(* CoDeSys 2.3.9.41 project: fongus.pro *)
(* Libraries: STANDARD.LIB 4.10.05 11:14:46, IECSFC.LIB 13.4.06 15:51:28, ANALYZATION.LIB 5.10.99 09:05:06 *)

(* PLC configuration (modules and I/O channels)
DI0_staticRun AT %IX0.0 [BitInput]
DI1_dynamicRun AT %IX0.1 [BitInput]
AT %IX0.2 [BitInput]
AT %IX0.3 [BitInput]
AT %IX0.4 [BitInput]
AT %IX0.5 [BitInput]
DO0_filter AT %QX1.0 [BitOutput]
AT %QX1.1 [BitOutput]
AT %QX1.2 [BitOutput]
AT %QX1.3 [BitOutput]
Special output [ID104] node 2, in %IB2 out %QB2 {Visibility = No; PinCount = 1}
  AT %QX2.0 [BitOutput] Special output
Unifed signal sensor [ID700] node 3, in %IB3 out %QB3 {Type_of_sensor700 = IT_0_20; measure_interval = 0.8; ainlow = 0; ainhigh = 20; first_cor_point = 0; first_delta = 0; second_cor_point = 0; second_delta = 0; third_cor_point = 0; third_delta = 0; Visibility = No}
  AT %ID3.0 [FloatInput] Value
  AT %IW3.1 [WordInput] Circular time
  Analog Input [ID107] node 0, in %IB3.0 out %QB3.0
Unifed signal sensor [ID700] node 4, in %IB4 out %QB4 {Type_of_sensor700 = IT_0_20; measure_interval = 0.8; ainlow = 0; ainhigh = 20; first_cor_point = 0; first_delta = 0; second_cor_point = 0; second_delta = 0; third_cor_point = 0; third_delta = 0; Visibility = No}
  AT %ID4.0 [FloatInput] Value
  AT %IW4.1 [WordInput] Circular time
  Analog Input [ID107] node 0, in %IB4.0 out %QB4.0
Unifed signal sensor [ID700] node 5, in %IB5 out %QB5 {Type_of_sensor700 = IT_0_20; measure_interval = 0.8; ainlow = 0; ainhigh = 20; first_cor_point = 0; first_delta = 0; second_cor_point = 0; second_delta = 0; third_cor_point = 0; third_delta = 0; Visibility = No}
  AT %ID5.0 [FloatInput] Value
  AT %IW5.1 [WordInput] Circular time
  Analog Input [ID107] node 0, in %IB5.0 out %QB5.0
Unifed signal sensor [ID700] node 6, in %IB6 out %QB6 {Type_of_sensor700 = IT_0_20; measure_interval = 0.8; ainlow = 0; ainhigh = 20; first_cor_point = 0; first_delta = 0; second_cor_point = 0; second_delta = 0; third_cor_point = 0; third_delta = 0; Visibility = No}
  AT %ID6.0 [FloatInput] Value
  AT %IW6.1 [WordInput] Circular time
  Analog Input [ID107] node 0, in %IB6.0 out %QB6.0
AO0_fc1 AT %QD7.0 [FloatOutput] Value
AO1_fc2 AT %QD8.0 [FloatOutput] Value
Modbus [MODBUS_ID302] node 0, in %IB9.0 out %QB9.0
  Debug RS-232 [DEBUG_USART] node 0, in %IB9.0.0 out %QB9.0.0 {CommunicationSpeed = 11520; Parity = NO PARITY CHECK; BitLength = 8 bits; StopLength = One stop bit; InterfaceType = RS232; FrameOriented = ASCII; Timeout = 0; Visibility = No}
pan_BITS0 AT %QW9.1.0 [WordOutput] man
pan_BITS1 AT %QW9.2.0 [WordOutput]
pan_BITS2 AT %QW9.3.0 [WordOutput]
pan_BITS3 AT %QW9.4.0 [WordOutput]
2 byte [Register] node 5, in %IB9.5 out %QB9.5
  fc1_p1t AT %QW9.5.0 [WordOutput]
2 byte [Register] node 6, in %IB9.6 out %QB9.6
  fc1_p2t AT %QW9.6.0 [WordOutput]
2 byte [Register] node 7, in %IB9.7 out %QB9.7
  fc1_p3t AT %QW9.7.0 [WordOutput]
2 byte [Register] node 8, in %IB9.8 out %QB9.8
  fc1_p4t AT %QW9.8.0 [WordOutput]
2 byte [Register] node 9, in %IB9.9 out %QB9.9
  fc1_p5t AT %QW9.9.0 [WordOutput]
2 byte [Register] node 10, in %IB9.10 out %QB9.10
  fc1_p6t AT %QW9.10.0 [WordOutput]
2 byte [Register] node 11, in %IB9.11 out %QB9.11
  fc1_p7t AT %QW9.11.0 [WordOutput]
2 byte [Register] node 12, in %IB9.12 out %QB9.12
  fc1_p8t AT %QW9.12.0 [WordOutput]
2 byte [Register] node 13, in %IB9.13 out %QB9.13
  fc1_p9t AT %QW9.13.0 [WordOutput]
2 byte [Register] node 14, in %IB9.14 out %QB9.14
  fc1_p10t AT %QW9.14.0 [WordOutput]
2 byte [Register] node 15, in %IB9.15 out %QB9.15
  fc1_p1v AT %QW9.15.0 [WordOutput]
2 byte [Register] node 16, in %IB9.16 out %QB9.16
  fc1_p2v AT %QW9.16.0 [WordOutput]
2 byte [Register] node 17, in %IB9.17 out %QB9.17
  fc1_p3v AT %QW9.17.0 [WordOutput]
2 byte [Register] node 18, in %IB9.18 out %QB9.18
  fc1_p4v AT %QW9.18.0 [WordOutput]
2 byte [Register] node 19, in %IB9.19 out %QB9.19
  fc1_p5v AT %QW9.19.0 [WordOutput]
2 byte [Register] node 20, in %IB9.20 out %QB9.20
  fc1_p6v AT %QW9.20.0 [WordOutput]
2 byte [Register] node 21, in %IB9.21 out %QB9.21
  fc1_p7v AT %QW9.21.0 [WordOutput]
2 byte [Register] node 22, in %IB9.22 out %QB9.22
  fc1_p8v AT %QW9.22.0 [WordOutput]
2 byte [Register] node 23, in %IB9.23 out %QB9.23
  fc1_p9v AT %QW9.23.0 [WordOutput]
2 byte [Register] node 24, in %IB9.24 out %QB9.24
  fc1_p10v AT %QW9.24.0 [WordOutput]
2 byte [Register] node 25, in %IB9.25 out %QB9.25
  fc2_p1t AT %QW9.25.0 [WordOutput]
2 byte [Register] node 26, in %IB9.26 out %QB9.26
  fc2_p2t AT %QW9.26.0 [WordOutput]
2 byte [Register] node 27, in %IB9.27 out %QB9.27
  fc2_p3t AT %QW9.27.0 [WordOutput]
2 byte [Register] node 28, in %IB9.28 out %QB9.28
  fc2_p4t AT %QW9.28.0 [WordOutput]
2 byte [Register] node 29, in %IB9.29 out %QB9.29
  fc2_p5t AT %QW9.29.0 [WordOutput]
2 byte [Register] node 30, in %IB9.30 out %QB9.30
  fc2_p6t AT %QW9.30.0 [WordOutput]
2 byte [Register] node 31, in %IB9.31 out %QB9.31
  fc2_p7t AT %QW9.31.0 [WordOutput]
2 byte [Register] node 32, in %IB9.32 out %QB9.32
  fc2_p8t AT %QW9.32.0 [WordOutput]
2 byte [Register] node 33, in %IB9.33 out %QB9.33
  fc2_p9t AT %QW9.33.0 [WordOutput]
2 byte [Register] node 34, in %IB9.34 out %QB9.34
  fc2_p10t AT %QW9.34.0 [WordOutput]
2 byte [Register] node 35, in %IB9.35 out %QB9.35
  fc2_p1v AT %QW9.35.0 [WordOutput]
2 byte [Register] node 36, in %IB9.36 out %QB9.36
  fc2_p2v AT %QW9.36.0 [WordOutput]
2 byte [Register] node 37, in %IB9.37 out %QB9.37
  fc2_p3v AT %QW9.37.0 [WordOutput]
2 byte [Register] node 38, in %IB9.38 out %QB9.38
  fc2_p4v AT %QW9.38.0 [WordOutput]
2 byte [Register] node 39, in %IB9.39 out %QB9.39
  fc2_p5v AT %QW9.39.0 [WordOutput]
2 byte [Register] node 40, in %IB9.40 out %QB9.40
  fc2_p6v AT %QW9.40.0 [WordOutput]
2 byte [Register] node 41, in %IB9.41 out %QB9.41
  fc2_p7v AT %QW9.41.0 [WordOutput]
2 byte [Register] node 42, in %IB9.42 out %QB9.42
  fc2_p8v AT %QW9.42.0 [WordOutput]
2 byte [Register] node 43, in %IB9.43 out %QB9.43
  fc2_p9v AT %QW9.43.0 [WordOutput]
2 byte [Register] node 44, in %IB9.44 out %QB9.44
  fc2_p10v AT %QW9.44.0 [WordOutput]
2 byte [Register] node 45, in %IB9.45 out %QB9.45
  fc1_staticValue AT %QW9.45.0 [WordOutput]
  fc2_staticValue AT %QW9.46.0 [WordOutput]
  pan_evilStartHH AT %QW9.47.0 [WordOutput]
  pan_evilStartMM AT %QW9.48.0 [WordOutput]
  pan_evilStopHH AT %QW9.49.0 [WordOutput]
  pan_evilStopMM AT %QW9.50.0 [WordOutput]
  pan_holyStartHH AT %QW9.51.0 [WordOutput]
  pan_holyStartMM AT %QW9.52.0 [WordOutput]
  pan_holyStopHH AT %QW9.53.0 [WordOutput]
  pan_holyStopMM AT %QW9.54.0 [WordOutput]
  pan_EVILDAYS AT %QW9.55.0 [WordOutput]
  pan_HOLYDAYS AT %QW9.56.0 [WordOutput]
  pan_fe1_onHH AT %QW9.57.0 [WordOutput]
  pan_fe1_onMM AT %QW9.58.0 [WordOutput]
  pan_fe1_offHH AT %QW9.59.0 [WordOutput]
  pan_fe1_offMM AT %QW9.60.0 [WordOutput]
  pan_fe2_onHH AT %QW9.61.0 [WordOutput]
  pan_fe2_onMM AT %QW9.62.0 [WordOutput]
  pan_fe2_offHH AT %QW9.63.0 [WordOutput]
  pan_fe2_offMM AT %QW9.64.0 [WordOutput]
  pan_fe3_onHH AT %QW9.65.0 [WordOutput]
  pan_fe3_onMM AT %QW9.66.0 [WordOutput]
  pan_fe3_offHH AT %QW9.67.0 [WordOutput]
  pan_fe3_offMM AT %QW9.68.0 [WordOutput]
  pan_fe4_onHH AT %QW9.69.0 [WordOutput]
  pan_fe4_onMM AT %QW9.70.0 [WordOutput]
  pan_fe4_offHH AT %QW9.71.0 [WordOutput]
  pan_fe4_offMM AT %QW9.72.0 [WordOutput]
  pan_fe5_onHH AT %QW9.73.0 [WordOutput]
  pan_fe5_onMM AT %QW9.74.0 [WordOutput]
  pan_fe5_offHH AT %QW9.75.0 [WordOutput]
  pan_fe5_offMM AT %QW9.76.0 [WordOutput]
  pan_fe6_onHH AT %QW9.77.0 [WordOutput]
  pan_fe6_onMM AT %QW9.78.0 [WordOutput]
  pan_fe6_offHH AT %QW9.79.0 [WordOutput]
  pan_fe6_offMM AT %QW9.80.0 [WordOutput]
*)

(* Global variable list: Global_Variables *)
VAR_GLOBAL

(* Times *)
	GetTime: CurTimeEx;
	TimeAndDate: SystemTimeDate;
	Sys_Time: SysTime64;

END_VAR

(* POU PLC_PRG, ST *)
PROGRAM PLC_PRG
VAR
	setYear : INT;
	setMonth, setDay, setHour, setMinute : BYTE;
	set_time : BOOL;
END_VAR

END_PROGRAM
ACTION Times:
TimeAndDate.Day :=0;
TimeAndDate.DayOfWeek :=0;
TimeAndDate.dwHighMsec :=0;
TimeAndDate.dwLowMSecs :=0;
TimeAndDate.Milliseconds :=0;
TimeAndDate.Minute :=0;
TimeAndDate.Second :=0;
TimeAndDate.Hour :=0;
TimeAndDate.Year :=0;
TimeAndDate.Month :=0;
Sys_time.ulHigh :=0;
Sys_time.ulLow :=0;
GetTime (SystemTime:=Sys_Time , TimeDate:= TimeAndDate);


IF set_time THEN

	TimeAndDate.Minute:=setMinute;
	TimeAndDate.Second:=0;
	TimeAndDate.Hour:=setHour;
	TimeAndDate.Day:=setDay;
	TimeAndDate.Month:=setMonth;
	TimeAndDate.Year:=setYear;
	GetTime (SystemTime:=Sys_Time , TimeDate:= TimeAndDate);

END_IF
END_ACTION

(* POU FOUNTAIN, ST *)
PROGRAM FOUNTAIN
VAR
	start : BOOL;
	startByDays : BOOL;
	dynamic, static : BOOL;
	evilStartHH, evilStartMM, evilStopHH, evilStopMM : WORD;
	holyStartHH, holyStartMM, holyStopHH, holyStopMM : WORD;

	(* filter *)
	 filterRun, filterSchedGo : BOOL;
	fe1, fe2, fe3, fe4, fe5, fe6 : TimeOnCheck;
	fe1state, fe2state, fe3state, fe4state, fe5state, fe6state : BOOL;

	(* days *)
	evilTimeCheck, holyTimeCheck : TimeOnCheck;
	evilDayOk, holyDayOk : BOOL;

	M1, N1 : BOOL;
	founT1, founTN1 : TON;
	M2, N2 : BOOL;
	founT2, founTN2 : TON;
	M3, N3 : BOOL;
	founT3, founTN3 : TON;
	M4, N4 : BOOL;
	founT4, founTN4 : TON;
	M5, N5 : BOOL;
	founT5, founTN5 : TON;
	M6, N6 : BOOL;
	founT6, founTN6 : TON;
	M7, N7 : BOOL;
	founT7, founTN7 : TON;
	M8, N8 : BOOL;
	founT8, founTN8 : TON;
	M9, N9 : BOOL;
	founT9, founTN9 : TON;
	M10, N10 : BOOL;
	founT10, founTN10 : TON;

	FPFON: R_TRIG;
	FPFONN : R_TRIG;

	(*galetMode : BOOL;*)

END_VAR

VAR RETAIN
	(* filter *)
	filterMan, filterAuto : BOOL;
	fe1_onHH, fe1_onMM, fe1_offHH, fe1_offMM : WORD;
	fe2_onHH, fe2_onMM, fe2_offHH, fe2_offMM : WORD;
	fe3_onHH, fe3_onMM, fe3_offHH, fe3_offMM : WORD;
	fe4_onHH, fe4_onMM, fe4_offHH, fe4_offMM : WORD;
	fe5_onHH, fe5_onMM, fe5_offHH, fe5_offMM : WORD;
	fe6_onHH, fe6_onMM, fe6_offHH, fe6_offMM : WORD;

	staticFValue : REAL;
	staticFValueN : REAL;
	EVILDAYS, HOLYDAYS : WORD;

	(* fc1 *)
	founV1F: REAL;
	founV2F: REAL;
	founV3F: REAL;
	founV4F: REAL;
	founV5F: REAL;
	founV6F: REAL;
	founV7F: REAL;
	founV8F: REAL;
	founV9F: REAL;
	founV10F: REAL;

	founS1T: TIME;
	founS2T: TIME;
	founS3T: TIME;
	founS4T: TIME;
	founS5T: TIME;
	founS6T: TIME;
	founS7T: TIME;
	founS8T: TIME;
	founS9T: TIME;
	founS10T: TIME;

(* fc2 *)
	founV1FN: REAL;
	founV2FN: REAL;
	founV3FN: REAL;
	founV4FN: REAL;
	founV5FN: REAL;
	founV6FN: REAL;
	founV7FN: REAL;
	founV8FN: REAL;
	founV9FN: REAL;
	founV10FN: REAL;

	founS1TN: TIME;
	founS2TN: TIME;
	founS3TN: TIME;
	founS4TN: TIME;
	founS5TN: TIME;
	founS6TN: TIME;
	founS7TN: TIME;
	founS8TN: TIME;
	founS9TN: TIME;
	founS10TN: TIME;

(* days *)
	evilStartHH, evilStartMM, evilStopHH, evitStopMM : WORD;
	holyStartHH, holyStartMM, holyStopHH, holyStopMM : WORD;
END_VAR
VAR (* helpers for the ST form of the networks *)
	_p1 : BOOL;
	_p2 : BOOL;
	_p3 : BOOL;
	_p4 : BOOL;
	_p5 : BOOL;
	_p6 : BOOL;
	_p7 : BOOL;
	_p8 : BOOL;
	_p9 : BOOL;
	_p10 : BOOL;
	_p11 : BOOL;
	_p12 : BOOL;
	_p13 : BOOL;
	_p14 : BOOL;
	_p15 : BOOL;
	_p16 : BOOL;
	_p17 : BOOL;
	_p18 : BOOL;
	_p19 : BOOL;
	_p20 : BOOL;
END_VAR
IF DI0_staticRun THEN
	static := TRUE;
ELSE
	static := FALSE;
END_IF;

IF DI1_dynamicRun THEN
	dynamic := TRUE;
ELSE
	dynamic := FALSE;
END_IF;


IF ( founV1F = 0.0 ) AND
	( founV2F = 0.0 ) AND
	( founV3F = 0.0 ) AND
	( founV4F = 0.0 ) AND
	( founV5F = 0.0 ) AND
	( founV6F = 0.0 ) AND
	( founV7F = 0.0 ) AND
	( founV8F = 0.0 ) AND
	( founV9F = 0.0 ) AND
	( founV10F = 0.0 )
THEN
	(*nodyn := TRUE;*)
END_IF;

IF startByDays THEN
	start := TRUE;
ELSE
	start := FALSE;
END_IF;

IF start THEN
	AOvalues;
	AONvalues;
ELSE
	AO0_fc1 := 0.0;
	AO1_fc2 := 0.0;
END_IF;
END_PROGRAM
ACTION AONvalues:
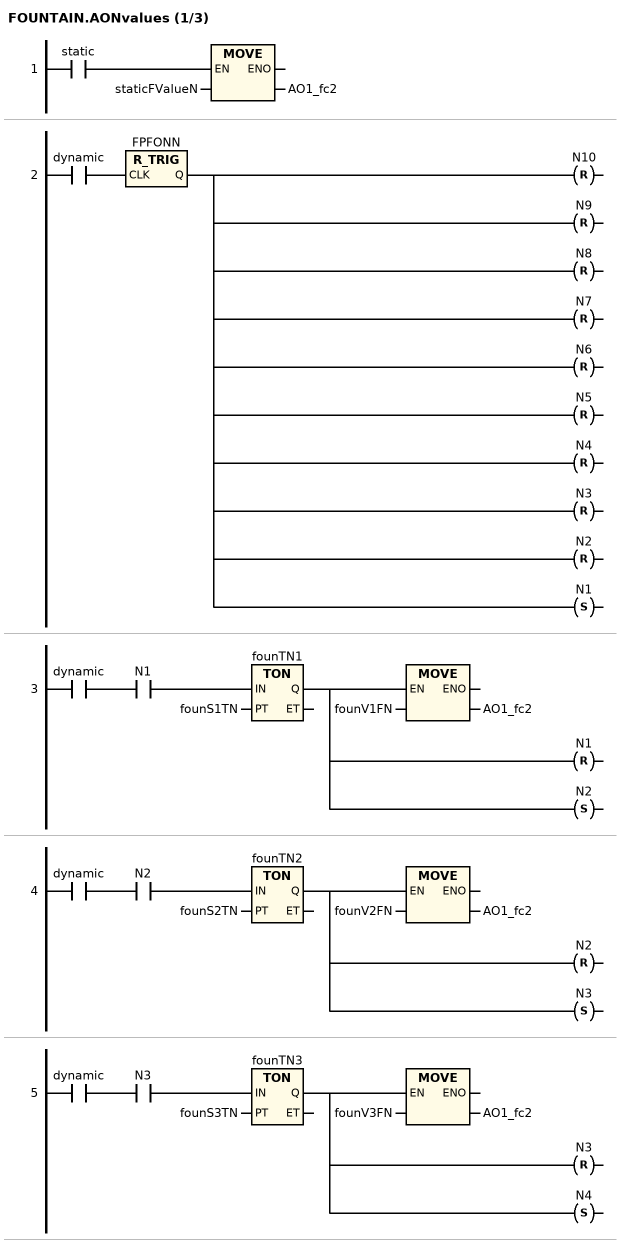
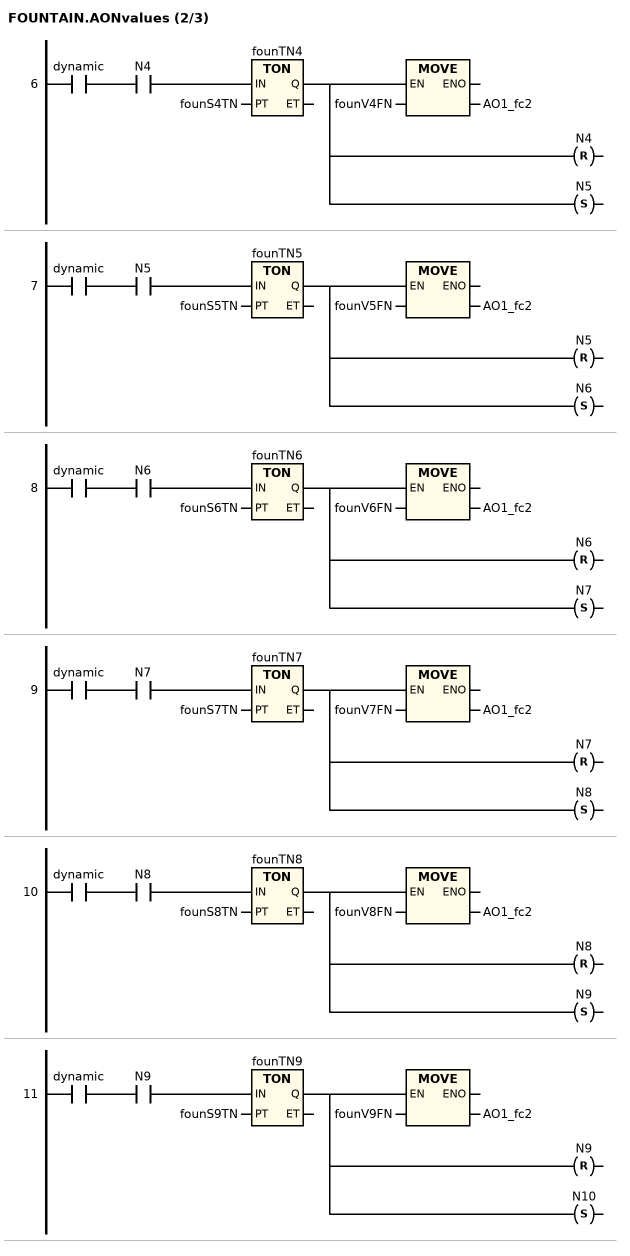
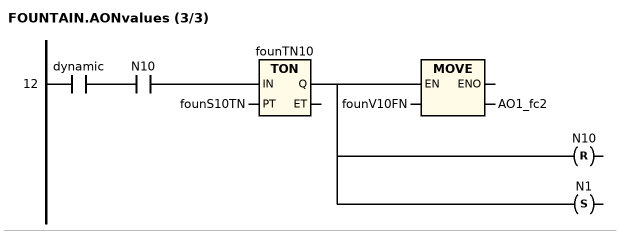
_LD_ (* Ladder Diagram *)
NETWORK 1
	[static]
		EN --- MOVE(staticFValueN) => AO1_fc2
NETWORK 2
	[dynamic] - FPFONN:R_TRIG(CLK: *) --- (R N10) (R N9) (R N8) (R N7) (R N6) (R N5) (R N4) (R N3) (R N2) (S N1)
NETWORK 3
	[dynamic] - [N1] - founTN1:TON(IN: *, PT: founS1TN) --- (R N1) (S N2)
		EN --- MOVE(founV1FN) => AO1_fc2
NETWORK 4
	[dynamic] - [N2] - founTN2:TON(IN: *, PT: founS2TN) --- (R N2) (S N3)
		EN --- MOVE(founV2FN) => AO1_fc2
NETWORK 5
	[dynamic] - [N3] - founTN3:TON(IN: *, PT: founS3TN) --- (R N3) (S N4)
		EN --- MOVE(founV3FN) => AO1_fc2
NETWORK 6
	[dynamic] - [N4] - founTN4:TON(IN: *, PT: founS4TN) --- (R N4) (S N5)
		EN --- MOVE(founV4FN) => AO1_fc2
NETWORK 7
	[dynamic] - [N5] - founTN5:TON(IN: *, PT: founS5TN) --- (R N5) (S N6)
		EN --- MOVE(founV5FN) => AO1_fc2
NETWORK 8
	[dynamic] - [N6] - founTN6:TON(IN: *, PT: founS6TN) --- (R N6) (S N7)
		EN --- MOVE(founV6FN) => AO1_fc2
NETWORK 9
	[dynamic] - [N7] - founTN7:TON(IN: *, PT: founS7TN) --- (R N7) (S N8)
		EN --- MOVE(founV7FN) => AO1_fc2
NETWORK 10
	[dynamic] - [N8] - founTN8:TON(IN: *, PT: founS8TN) --- (R N8) (S N9)
		EN --- MOVE(founV8FN) => AO1_fc2
NETWORK 11
	[dynamic] - [N9] - founTN9:TON(IN: *, PT: founS9TN) --- (R N9) (S N10)
		EN --- MOVE(founV9FN) => AO1_fc2
NETWORK 12
	[dynamic] - [N10] - founTN10:TON(IN: *, PT: founS10TN) --- (R N10) (S N1)
		EN --- MOVE(founV10FN) => AO1_fc2
_END_LD_
(* the same logic as Structured Text *)
(* Network 1 *)
IF static THEN
	AO1_fc2 := staticFValueN;
END_IF;
(* Network 2 *)
FPFONN(CLK := dynamic);
IF FPFONN.Q THEN N10 := FALSE; N9 := FALSE; N8 := FALSE; N7 := FALSE; N6 := FALSE; N5 := FALSE; N4 := FALSE; N3 := FALSE; N2 := FALSE; N1 := TRUE; END_IF;
(* Network 3 *)
founTN1(IN := dynamic AND N1, PT := founS1TN);
_p1 := founTN1.Q;
IF _p1 THEN
	AO1_fc2 := founV1FN;
END_IF;
IF _p1 THEN N1 := FALSE; N2 := TRUE; END_IF;
(* Network 4 *)
founTN2(IN := dynamic AND N2, PT := founS2TN);
_p2 := founTN2.Q;
IF _p2 THEN
	AO1_fc2 := founV2FN;
END_IF;
IF _p2 THEN N2 := FALSE; N3 := TRUE; END_IF;
(* Network 5 *)
founTN3(IN := dynamic AND N3, PT := founS3TN);
_p3 := founTN3.Q;
IF _p3 THEN
	AO1_fc2 := founV3FN;
END_IF;
IF _p3 THEN N3 := FALSE; N4 := TRUE; END_IF;
(* Network 6 *)
founTN4(IN := dynamic AND N4, PT := founS4TN);
_p4 := founTN4.Q;
IF _p4 THEN
	AO1_fc2 := founV4FN;
END_IF;
IF _p4 THEN N4 := FALSE; N5 := TRUE; END_IF;
(* Network 7 *)
founTN5(IN := dynamic AND N5, PT := founS5TN);
_p5 := founTN5.Q;
IF _p5 THEN
	AO1_fc2 := founV5FN;
END_IF;
IF _p5 THEN N5 := FALSE; N6 := TRUE; END_IF;
(* Network 8 *)
founTN6(IN := dynamic AND N6, PT := founS6TN);
_p6 := founTN6.Q;
IF _p6 THEN
	AO1_fc2 := founV6FN;
END_IF;
IF _p6 THEN N6 := FALSE; N7 := TRUE; END_IF;
(* Network 9 *)
founTN7(IN := dynamic AND N7, PT := founS7TN);
_p7 := founTN7.Q;
IF _p7 THEN
	AO1_fc2 := founV7FN;
END_IF;
IF _p7 THEN N7 := FALSE; N8 := TRUE; END_IF;
(* Network 10 *)
founTN8(IN := dynamic AND N8, PT := founS8TN);
_p8 := founTN8.Q;
IF _p8 THEN
	AO1_fc2 := founV8FN;
END_IF;
IF _p8 THEN N8 := FALSE; N9 := TRUE; END_IF;
(* Network 11 *)
founTN9(IN := dynamic AND N9, PT := founS9TN);
_p9 := founTN9.Q;
IF _p9 THEN
	AO1_fc2 := founV9FN;
END_IF;
IF _p9 THEN N9 := FALSE; N10 := TRUE; END_IF;
(* Network 12 *)
founTN10(IN := dynamic AND N10, PT := founS10TN);
_p10 := founTN10.Q;
IF _p10 THEN
	AO1_fc2 := founV10FN;
END_IF;
IF _p10 THEN N10 := FALSE; N1 := TRUE; END_IF;
END_ACTION
ACTION AOvalues:
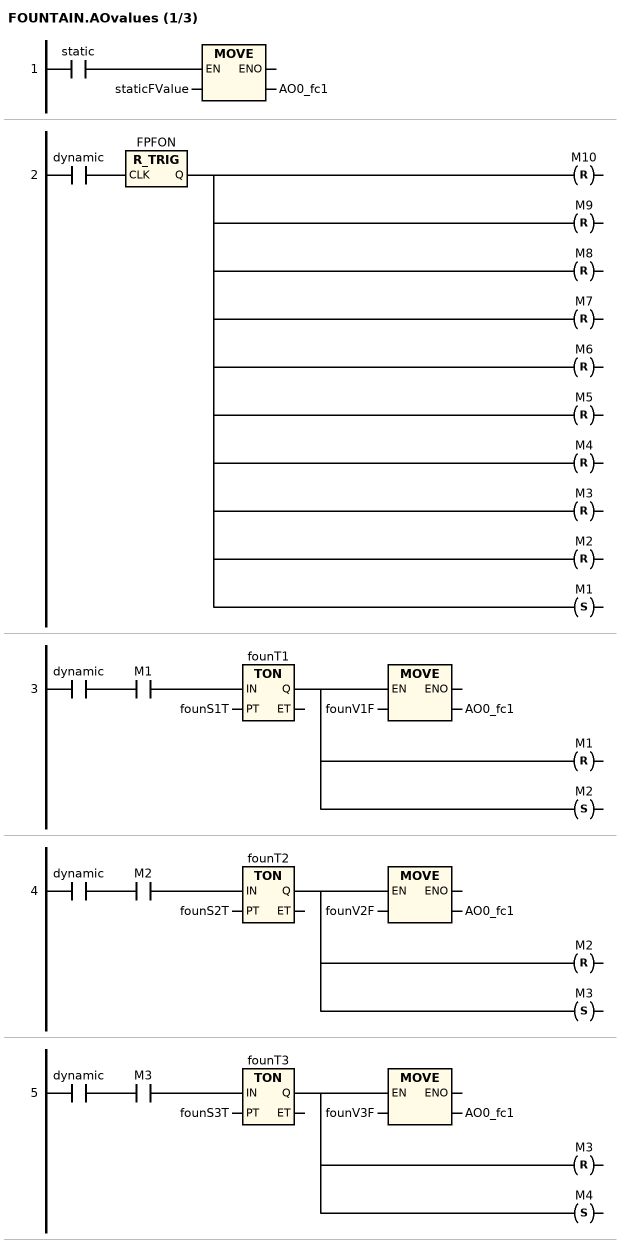
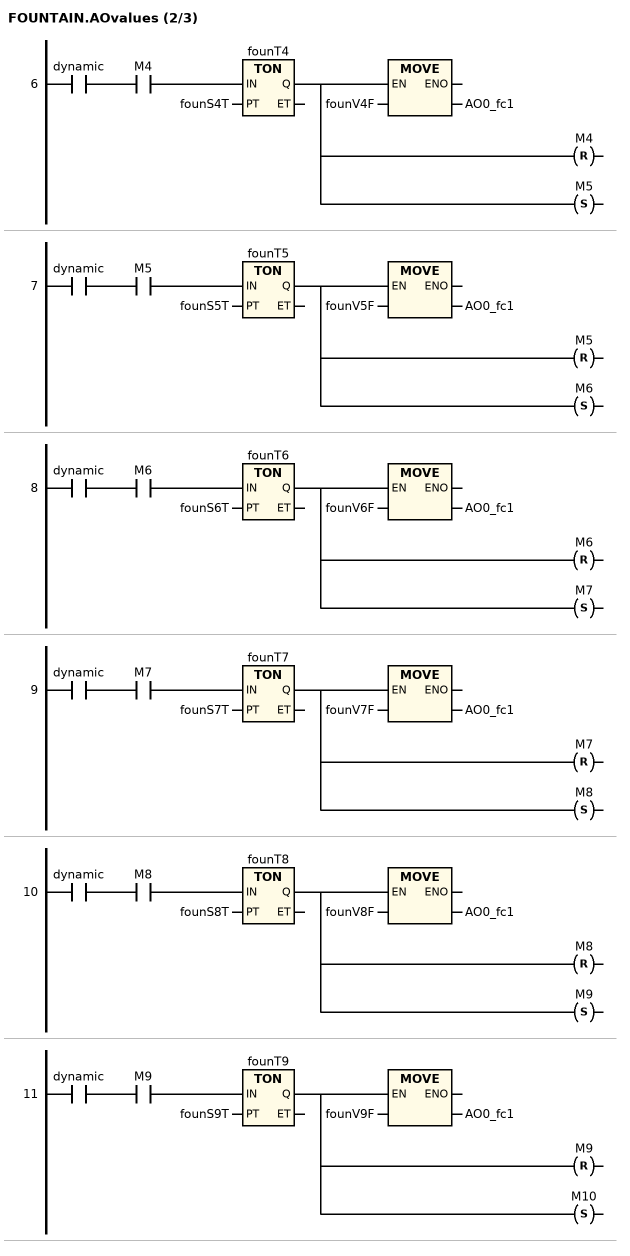
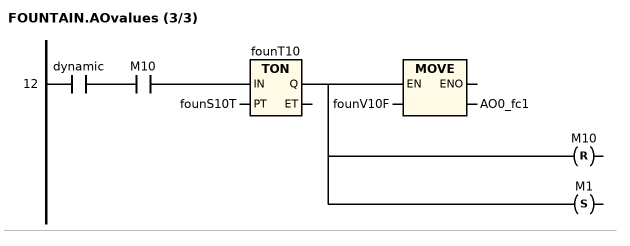
_LD_ (* Ladder Diagram *)
NETWORK 1
	[static]
		EN --- MOVE(staticFValue) => AO0_fc1
NETWORK 2
	[dynamic] - FPFON:R_TRIG(CLK: *) --- (R M10) (R M9) (R M8) (R M7) (R M6) (R M5) (R M4) (R M3) (R M2) (S M1)
NETWORK 3
	[dynamic] - [M1] - founT1:TON(IN: *, PT: founS1T) --- (R M1) (S M2)
		EN --- MOVE(founV1F) => AO0_fc1
NETWORK 4
	[dynamic] - [M2] - founT2:TON(IN: *, PT: founS2T) --- (R M2) (S M3)
		EN --- MOVE(founV2F) => AO0_fc1
NETWORK 5
	[dynamic] - [M3] - founT3:TON(IN: *, PT: founS3T) --- (R M3) (S M4)
		EN --- MOVE(founV3F) => AO0_fc1
NETWORK 6
	[dynamic] - [M4] - founT4:TON(IN: *, PT: founS4T) --- (R M4) (S M5)
		EN --- MOVE(founV4F) => AO0_fc1
NETWORK 7
	[dynamic] - [M5] - founT5:TON(IN: *, PT: founS5T) --- (R M5) (S M6)
		EN --- MOVE(founV5F) => AO0_fc1
NETWORK 8
	[dynamic] - [M6] - founT6:TON(IN: *, PT: founS6T) --- (R M6) (S M7)
		EN --- MOVE(founV6F) => AO0_fc1
NETWORK 9
	[dynamic] - [M7] - founT7:TON(IN: *, PT: founS7T) --- (R M7) (S M8)
		EN --- MOVE(founV7F) => AO0_fc1
NETWORK 10
	[dynamic] - [M8] - founT8:TON(IN: *, PT: founS8T) --- (R M8) (S M9)
		EN --- MOVE(founV8F) => AO0_fc1
NETWORK 11
	[dynamic] - [M9] - founT9:TON(IN: *, PT: founS9T) --- (R M9) (S M10)
		EN --- MOVE(founV9F) => AO0_fc1
NETWORK 12
	[dynamic] - [M10] - founT10:TON(IN: *, PT: founS10T) --- (R M10) (S M1)
		EN --- MOVE(founV10F) => AO0_fc1
_END_LD_
(* the same logic as Structured Text *)
(* Network 1 *)
IF static THEN
	AO0_fc1 := staticFValue;
END_IF;
(* Network 2 *)
FPFON(CLK := dynamic);
IF FPFON.Q THEN M10 := FALSE; M9 := FALSE; M8 := FALSE; M7 := FALSE; M6 := FALSE; M5 := FALSE; M4 := FALSE; M3 := FALSE; M2 := FALSE; M1 := TRUE; END_IF;
(* Network 3 *)
founT1(IN := dynamic AND M1, PT := founS1T);
_p11 := founT1.Q;
IF _p11 THEN
	AO0_fc1 := founV1F;
END_IF;
IF _p11 THEN M1 := FALSE; M2 := TRUE; END_IF;
(* Network 4 *)
founT2(IN := dynamic AND M2, PT := founS2T);
_p12 := founT2.Q;
IF _p12 THEN
	AO0_fc1 := founV2F;
END_IF;
IF _p12 THEN M2 := FALSE; M3 := TRUE; END_IF;
(* Network 5 *)
founT3(IN := dynamic AND M3, PT := founS3T);
_p13 := founT3.Q;
IF _p13 THEN
	AO0_fc1 := founV3F;
END_IF;
IF _p13 THEN M3 := FALSE; M4 := TRUE; END_IF;
(* Network 6 *)
founT4(IN := dynamic AND M4, PT := founS4T);
_p14 := founT4.Q;
IF _p14 THEN
	AO0_fc1 := founV4F;
END_IF;
IF _p14 THEN M4 := FALSE; M5 := TRUE; END_IF;
(* Network 7 *)
founT5(IN := dynamic AND M5, PT := founS5T);
_p15 := founT5.Q;
IF _p15 THEN
	AO0_fc1 := founV5F;
END_IF;
IF _p15 THEN M5 := FALSE; M6 := TRUE; END_IF;
(* Network 8 *)
founT6(IN := dynamic AND M6, PT := founS6T);
_p16 := founT6.Q;
IF _p16 THEN
	AO0_fc1 := founV6F;
END_IF;
IF _p16 THEN M6 := FALSE; M7 := TRUE; END_IF;
(* Network 9 *)
founT7(IN := dynamic AND M7, PT := founS7T);
_p17 := founT7.Q;
IF _p17 THEN
	AO0_fc1 := founV7F;
END_IF;
IF _p17 THEN M7 := FALSE; M8 := TRUE; END_IF;
(* Network 10 *)
founT8(IN := dynamic AND M8, PT := founS8T);
_p18 := founT8.Q;
IF _p18 THEN
	AO0_fc1 := founV8F;
END_IF;
IF _p18 THEN M8 := FALSE; M9 := TRUE; END_IF;
(* Network 11 *)
founT9(IN := dynamic AND M9, PT := founS9T);
_p19 := founT9.Q;
IF _p19 THEN
	AO0_fc1 := founV9F;
END_IF;
IF _p19 THEN M9 := FALSE; M10 := TRUE; END_IF;
(* Network 12 *)
founT10(IN := dynamic AND M10, PT := founS10T);
_p20 := founT10.Q;
IF _p20 THEN
	AO0_fc1 := founV10F;
END_IF;
IF _p20 THEN M10 := FALSE; M1 := TRUE; END_IF;
END_ACTION
ACTION Days:
CASE TimeAndDate.DayOfWeek OF
	1 : IF EVILDAYS.1
	     	THEN evilDayOk := TRUE;
		ELSE evilDayOk := FALSE;
	     END_IF;

	2 : IF EVILDAYS.2
	     	THEN evilDayOk := TRUE;
		ELSE evilDayOk := FALSE;
	     END_IF;

      3 : IF EVILDAYS.3
	     	THEN evilDayOk := TRUE;
		ELSE evilDayOk := FALSE;
	     END_IF;

      4 : IF EVILDAYS.4
	     	THEN evilDayOk := TRUE;
		ELSE evilDayOk := FALSE;
	     END_IF;

      5 : IF EVILDAYS.5
	     	THEN evilDayOk := TRUE;
		ELSE evilDayOk := FALSE;
	     END_IF;

      6 : IF EVILDAYS.6
	     	THEN evilDayOk := TRUE;
		ELSE evilDayOk := FALSE;
	     END_IF;

      0 : IF EVILDAYS.0
	     	THEN evilDayOk := TRUE;
		ELSE evilDayOk := FALSE;
	     END_IF;
END_CASE;

CASE TimeAndDate.DayOfWeek OF
	1 : IF HOLYDAYS.1
	     	THEN holyDayOk := TRUE;
		ELSE holyDayOk := FALSE;
	     END_IF;

	2 : IF HOLYDAYS.2
	     	THEN holyDayOk := TRUE;
		ELSE holyDayOk := FALSE;
	     END_IF;

      3 : IF HOLYDAYS.3
	     	THEN holyDayOk := TRUE;
		ELSE holyDayOk := FALSE;
	     END_IF;

      4 : IF HOLYDAYS.4
	     	THEN holyDayOk := TRUE;
		ELSE holyDayOk := FALSE;
	     END_IF;

      5 : IF HOLYDAYS.5
	     	THEN holyDayOk := TRUE;
		ELSE holyDayOk := FALSE;
	     END_IF;

      6 : IF HOLYDAYS.6
	     	THEN holyDayOk := TRUE;
		ELSE holyDayOk := FALSE;
	     END_IF;

      0 : IF HOLYDAYS.0
	     	THEN holyDayOk := TRUE;
		ELSE holyDayOk := FALSE;
	     END_IF;
END_CASE;

IF evilDayOk THEN
	evilTimeCheck( currentState := startByDays,
					   needOffTime := TRUE,
					   onTime := 0, offTime := 0,
					    inonHH := evilStartHH,
					    inonMM := evilStartMM,
					    inoffHH := evilStopHH,
					    inoffMM := evilStopMM,
					    mustOn => startByDays );
ELSE
	IF holyDayOk THEN
		holyTimeCheck( currentState := startByDays,
					   needOffTime := TRUE,
					   onTime := 0, offTime := 0,
					    inonHH := holyStartHH,
					    inonMM := holyStartMM,
					    inoffHH := holyStopHH,
					    inoffMM := holyStopMM,
					    mustOn => startByDays );
	END_IF;
END_IF;
END_ACTION
ACTION Filter:
fe1 ( currentState := fe1state,
	   needOffTime := TRUE,
	   onTime := 0, offTime := 0,
	    inonHH := fe1_onHH,
	    inonMM := fe1_onMM,
	    inoffHH := fe1_offHH,
	    inoffMM := fe1_offMM,
	    mustOn => fe1state );


fe2 ( currentState := fe2state,
	   needOffTime := TRUE,
	   onTime := 0, offTime := 0,
	    inonHH := fe2_onHH,
	    inonMM := fe2_onMM,
	    inoffHH := fe2_offHH,
	    inoffMM := fe2_offMM,
	    mustOn => fe2state );


fe3 ( currentState := fe3state,
	   needOffTime := TRUE,
	   onTime := 0, offTime := 0,
	    inonHH := fe3_onHH,
	    inonMM := fe3_onMM,
	    inoffHH := fe3_offHH,
	    inoffMM := fe3_offMM,
	    mustOn => fe3state );



fe4 ( currentState := fe4state,
	   needOffTime := TRUE,
	   onTime := 0, offTime := 0,
	    inonHH := fe4_onHH,
	    inonMM := fe4_onMM,
	    inoffHH := fe4_offHH,
	    inoffMM := fe4_offMM,
	    mustOn => fe4state );


fe5 ( currentState := fe5state,
	   needOffTime := TRUE,
	   onTime := 0, offTime := 0,
	    inonHH := fe5_onHH,
	    inonMM := fe5_onMM,
	    inoffHH := fe5_offHH,
	    inoffMM := fe5_offMM,
	    mustOn => fe5state );


fe6 ( currentState := fe6state,
	   needOffTime := TRUE,
	   onTime := 0, offTime := 0,
	    inonHH := fe6_onHH,
	    inonMM := fe6_onMM,
	    inoffHH := fe6_offHH,
	    inoffMM := fe6_offMM,
	    mustOn => fe6state );

IF fe1state OR fe2state OR fe3state OR fe4state OR fe5state OR fe6state THEN
	filterSchedGo := TRUE;
ELSE
	filterSchedGo := FALSE;
END_IF;

IF filterMan OR ( filterAuto AND filterSchedGo ) THEN
	filterRun := TRUE;
ELSE
	filterRun := FALSE;
END_IF;
END_ACTION
ACTION Inputs:
(* filter *)
	fe1_onHH := pan_fe1_onHH;
	fe1_onMM := pan_fe1_onMM;
       fe1_offHH := pan_fe1_offHH;
	fe1_offMM := pan_fe1_offMM;
	fe2_onHH := pan_fe2_onHH;
	fe2_onMM := pan_fe2_onMM;
	fe2_offHH := pan_fe2_offHH;
	fe2_offMM := pan_fe2_offMM;
	fe3_onHH := pan_fe3_onHH;
	fe3_onMM := pan_fe3_onMM;
	fe3_offHH := pan_fe3_offHH;
	fe3_offMM := pan_fe3_offMM;
	fe4_onHH := pan_fe4_onHH;
	fe4_onMM := pan_fe4_onMM;
	fe4_offHH := pan_fe4_offHH;
	fe4_offMM := pan_fe4_offMM;
	fe5_onHH := pan_fe5_onHH;
	fe5_onMM := pan_fe5_onMM;
	fe5_offHH := pan_fe5_offHH
	fe5_offMM := pan_fe5_offMM;
	fe6_onHH := pan_fe6_onHH;
	fe6_onMM := pan_fe6_onMM;
	fe6_offHH := pan_fe6_offHH;
	fe6_offMM := pan_fe6_offMM;

(* days *)
	EVILDAYS := pan_EVILDAYS;
	HOLYDAYS := pan_HOLYDAYS;

	evilStartHH := pan_evilStartHH;
	evilStartMM := pan_evilStartMM;
	evilStopHH := pan_evilStopHH;
	evilStopMM := pan_evilStopMM;

	holyStartHH := pan_holyStartHH;
	holyStartMM := pan_holyStartMM;
	holyStopHH := pan_holyStopHH;
	holyStopMM := pan_holyStopMM;

(* fc1 *)
	staticFValue := WORD_TO_REAL ( fc1_staticValue );

	founV1F := WORD_TO_REAL( fc1_p1v );
	founV2F := WORD_TO_REAL( fc1_p2v );
	founV3F := WORD_TO_REAL( fc1_p3v );
	founV4F := WORD_TO_REAL( fc1_p4v );
	founV5F := WORD_TO_REAL( fc1_p5v );
	founV6F := WORD_TO_REAL( fc1_p6v );
	founV7F := WORD_TO_REAL( fc1_p7v );
	founV8F := WORD_TO_REAL( fc1_p8v );
	founV9F := WORD_TO_REAL( fc1_p9v );
	founV10F := WORD_TO_REAL( fc1_p10v );

	founS1T := WORD_TO_TIME ( fc1_p1t * 1000 );
	founS2T := WORD_TO_TIME ( fc1_p2t * 1000 );
	founS3T := WORD_TO_TIME ( fc1_p3t * 1000 );
	founS4T := WORD_TO_TIME ( fc1_p4t * 1000 );
	founS5T := WORD_TO_TIME ( fc1_p5t * 1000 );
	founS6T := WORD_TO_TIME ( fc1_p6t * 1000 );
	founS7T := WORD_TO_TIME ( fc1_p7t * 1000 );
	founS8T := WORD_TO_TIME ( fc1_p8t * 1000 );
	founS9T := WORD_TO_TIME ( fc1_p9t * 1000 );
	founS10T := WORD_TO_TIME ( fc1_p10t * 1000 );

(* fc2 *)
	staticFValueN := WORD_TO_REAL (  fc2_staticValue );

	founV1FN := WORD_TO_REAL( fc2_p1v );
	founV2FN := WORD_TO_REAL( fc2_p2v );
	founV3FN := WORD_TO_REAL( fc2_p3v );
	founV4FN := WORD_TO_REAL( fc2_p4v );
	founV5FN := WORD_TO_REAL( fc2_p5v );
	founV6FN := WORD_TO_REAL( fc2_p6v );
	founV7FN := WORD_TO_REAL( fc2_p7v );
	founV8FN := WORD_TO_REAL( fc2_p8v );
	founV9FN := WORD_TO_REAL( fc2_p9v );
	founV10FN := WORD_TO_REAL( fc2_p10v );

	founS1TN := WORD_TO_TIME ( fc2_p1t * 1000 );
	founS2TN := WORD_TO_TIME ( fc2_p2t * 1000 );
	founS3TN := WORD_TO_TIME ( fc2_p3t * 1000 );
	founS4TN := WORD_TO_TIME ( fc2_p4t * 1000 );
	founS5TN := WORD_TO_TIME ( fc2_p5t * 1000 );
	founS6TN := WORD_TO_TIME ( fc2_p6t * 1000 );
	founS7TN := WORD_TO_TIME ( fc2_p7t * 1000 );
	founS8TN := WORD_TO_TIME ( fc2_p8t * 1000 );
	founS9TN := WORD_TO_TIME ( fc2_p9t * 1000 );
	founS10TN := WORD_TO_TIME ( fc2_p10t * 1000 );
END_ACTION
ACTION Outputs:
DO0_filter := filterRun;
END_ACTION

(* POU TimeOnCheck, ST *)
FUNCTION_BLOCK TimeOnCheck
VAR_INPUT
	currentState : BOOL;
	needOffTime : BOOL;
	onTime : WORD;
	offTime : WORD;
	inonHH, inonMM : WORD;
	inoffHH, inoffMM : WORD;
END_VAR
VAR_OUTPUT
	mustOn : BOOL;
END_VAR
VAR
	onHH, onMM : BYTE;
	offHH, offMM : BYTE;
END_VAR
mustOn := currentState;

IF onTime <> 0 AND offTime <> 0 THEN
	onHH := WORD_TO_BYTE ( onTime );
	onMM := WORD_TO_BYTE ( onTime / 256 );

	offHH := WORD_TO_BYTE ( offTime );
	offMM := WORD_TO_BYTE ( offTime / 256 );
ELSE
	onHH := inonHH;
	onMM := inonMM;
	offHH := inonHH;
	offMM := inonMM;
END_IF;

IF needOffTime THEN
	IF onHH < offHH THEN
		IF ( onHH = offHH ) THEN
			IF ( onHH = TimeAndDate.Hour ) AND ( onMM <= TimeAndDate.Minute ) AND ( offMM > TimeAndDate.Minute ) THEN
				mustOn := TRUE;
			ELSE
				mustOn := FALSE;
			END_IF;
		ELSE
			IF ( onHH = TimeAndDate.Hour ) THEN
				IF ( onMM <= TimeAndDate.Minute ) THEN
					mustOn := TRUE;
				ELSE
					mustOn := FALSE;
				END_IF;
			ELSE
				IF ( onHH < TimeAndDate.Hour ) AND ( offHH > TimeAndDate.Hour ) THEN
					mustOn := TRUE;
				ELSE
					IF ( offHH = TimeAndDate.Hour ) THEN
						IF ( offMM > TimeAndDate.Minute ) THEN
							mustOn := TRUE;
						ELSE
							mustOn := FALSE;
						END_IF;
					ELSE
						mustOn := FALSE;
					END_IF;
				END_IF;
			END_IF;
		END_IF;
	ELSE (* onHH < offHH *)
		IF ( onHH = TimeAndDate.Hour ) THEN
			IF ( onMM <= TimeAndDate.Minute ) THEN
				mustOn := TRUE;
			ELSE
				mustOn := FALSE;
			END_IF;
		ELSE
			IF ( TimeAndDate.Hour > onHH ) AND ( TimeAndDate.Hour > offHH ) THEN
				mustOn := TRUE;
			ELSE
				IF ( TimeAndDate.Hour < offHH ) AND ( TimeAndDate.Hour < onHH ) THEN
					mustOn := TRUE;
				ELSE
					IF ( TimeAndDate.Hour = offHH ) THEN
						IF ( TimeAndDate.Minute < offMM ) THEN
							mustOn := TRUE;
						ELSE
							mustOn := FALSE;
						END_IF;
					ELSE
						mustOn := FALSE;
					END_IF;
				END_IF;
			END_IF;
		END_IF;
	END_IF; (* onHH < offHH *)
ELSE
	IF ( onHH = TimeAndDate.Hour ) AND ( onMM = TimeAndDate.Minute ) AND ( TimeAndDate.Second = 0 )
		THEN mustOn := TRUE;
	END_IF;
END_IF;
END_FUNCTION_BLOCK
